(* CODESYS project HomePLC_AlarmManager.library
   Company: Tom Oyen
   Description: Alarm manager
   Version: 1.0
   Placeholder: HomePLC Alarm Manager
   Author: Tom Oyen
   Title: HomePLC Alarm Manager

Project tree, tasks and I/O mapping:
  libraries: HomePLC DIO, * (Tom Oyen); HomePLC General, * (Tom Oyen); HomePLC Logging, * (Tom Oyen); Tc2_Standard, * (Beckhoff Automation GmbH); Tc2_System, * (Beckhoff Automation GmbH); Tc3_Module, * (Beckhoff Automation GmbH)
  DUTs/
    data type E_AlarmManagerStep
    data type E_AlarmState
    data type ST_AlarmManagerHMI
  GVLs/
    global variables GVL_AlarmManager
  POUs/
    Keypad/
      DUTs/
        data type E_KeypadState
        data type ST_AlarmKeypadHMI
        data type ST_AlarmKeypadVirtual
        data type ST_LedState
      function block FB_AlarmKeypad [ST]: CheckCode, CollectInput, Execute, FB_init, Reset, SetAlarmState, SetBuzzer, SetConfiguredCode, SetLeds, UpdateHMI, HmiData, Name
      interface I_AlarmKeypad: CheckCode, Execute, SetAlarmState, SetBuzzer, SetConfiguredCode, HmiData, Name
    Sensor/
      DUTs/
        data type ST_AlarmSensorHMI
      function block FB_AlarmSensor [ST]: Execute, FB_init, UpdateHMI, Alarm, AlarmTrigger, HmiData, Tamper, TamperTrigger, WarnFirst
      interface I_AlarmSensor: Execute, Alarm, AlarmTrigger, HmiData, Tamper, TamperTrigger, WarnFirst
    Siren/
      DUTs/
        data type ST_AlarmSirenHMI
      function block FB_AlarmSiren [ST]: Execute, FB_init, SetLight, SetSound, UpdateHMI, HmiData, Tamper, TamperTrigger
      interface I_AlarmSiren: Execute, SetLight, SetSound, HmiData, Tamper, TamperTrigger
    function block FB_AlarmManager [ST]: AddKeypad, AddSensor, AddSiren, Execute, Execute_Keypads, Execute_Sensors, Execute_Sirens, FB_init, UpdateHMI
    interface I_AlarmManager: AddKeypad, AddSensor, AddSiren
  Project Information/
    function F_GetCompany [ST]
    function F_GetTitle [ST]
    function F_GetVersion [ST]
  Version/
    global variables Global_Version
  VISUs/
    visualisation Alarm
    visualisation Keypad
    visualisation Sensor
    visualisation Siren
  text list GlobalTextList
*)

// DUTs/E_AlarmManagerStep
{attribute 'qualified_only'}
{attribute 'strict'}
TYPE E_AlarmManagerStep :
(
	Init 					:= 0,
	CheckEnable				:= 1,
	
	HardwareCheck			:= 10,
	Enabling				:= 11,
	Enable					:= 12,
	
	CheckSensors			:= 20,
	
	Warn					:= 30,
	WaitForDisableWarn		:= 31,
	SoundAlarm				:= 32,
	WaitForDisableAlarm		:= 33,
	
	DisableAlarm			:= 40,
	
	Reset					:= 50
);
END_TYPE

// DUTs/E_AlarmState
{attribute 'qualified_only'}
{attribute 'strict'}
TYPE E_AlarmState :
(
	Off 			:= 0,
	Enabling		:= 1,
	On				:= 2
);
END_TYPE

// DUTs/ST_AlarmManagerHMI
TYPE ST_AlarmManagerHMI :
STRUCT
	// General
	nKeypads	: INT;		// Number of keypads
	nSensors	: INT;		// Number of sensors
	nSirens		: INT;		// Number of sirens
	bEnabled	: BOOL;		// Alarm enabled state
	
	// Overview
	aSensors	: ARRAY [0..GVL_AlarmManager.nMaxSensors - 1] OF ST_AlarmSensorHMI;
	aSirens		: ARRAY [0..GVL_AlarmManager.nMaxSirens - 1] OF ST_AlarmSirenHMI;
END_STRUCT
END_TYPE

// POUs/Keypad/DUTs/E_KeypadState
{attribute 'qualified_only'}
{attribute 'strict'}
TYPE E_KeypadState :
(
	Init 				:= 0,
	Idle				:= 1,
	InputDetected		:= 2,
	CheckInput			:= 3,
	Reset				:= 4	
);
END_TYPE

// POUs/Keypad/DUTs/ST_AlarmKeypadHMI
TYPE ST_AlarmKeypadHMI :
STRUCT
	sName			: STRING;
	
	bLed1			: BOOL;
	bLed2			: BOOL;
	bLed3			: BOOL;
	bLed4			: BOOL;
	bLed5			: BOOL;
	bLed6			: BOOL;
	
	bBuzzer			: BOOL;
	
	sCode			: STRING;
END_STRUCT
END_TYPE

// POUs/Keypad/DUTs/ST_AlarmKeypadVirtual
TYPE ST_AlarmKeypadVirtual :
STRUCT
	bButton1			: BOOL;
	bButton2			: BOOL;
	bButton3			: BOOL;
	bButton4			: BOOL;
	bButton5			: BOOL;
	bButton6			: BOOL;
END_STRUCT
END_TYPE

// POUs/Keypad/DUTs/ST_LedState
TYPE ST_LedState :
STRUCT
	eLed1	: E_DOCommand;
	eLed2	: E_DOCommand;
	eLed3	: E_DOCommand;
	eLed4	: E_DOCommand;
	eLed5	: E_DOCommand;
	eLed6	: E_DOCommand;
END_STRUCT
END_TYPE

// POUs/Sensor/DUTs/ST_AlarmSensorHMI
TYPE ST_AlarmSensorHMI :
STRUCT
	sName		: STRING;	// Sensor name
	bAlarm		: BOOL;		// True if the sensor detects something
	bTamper		: BOOL;		// True if the sensor is tampered with
END_STRUCT
END_TYPE

// POUs/Siren/DUTs/ST_AlarmSirenHMI
TYPE ST_AlarmSirenHMI :
STRUCT
	sName		: STRING;	// Siren name
	bSiren		: BOOL;		// True if the siren is on
	bLight		: BOOL;		// True if the light is on
	bTamper		: BOOL;		// True if the siren is tampered with
END_STRUCT
END_TYPE

// GVLs/GVL_AlarmManager
{attribute 'qualified_only'}
VAR_GLOBAL CONSTANT
	nMaxKeypads		: INT := 5;										// Maximum number of keypads
	nMaxSirens		: INT := 5;										// Maximum number of sirens
	nMaxSensors		: INT := 10;									// Maximum number of sensors
	sCode			: STRING := '1234';								// Configured alarm code
END_VAR

// Version/Global_Version
{attribute 'TcGenerated'}
{attribute 'no-analysis'}
{attribute 'linkalways'}
// This function has been automatically generated from the project information.
VAR_GLOBAL CONSTANT
	{attribute 'const_non_replaced'}
	stLibVersion_HomePLC_Alarm_Manager : ST_LibVersion := (iMajor := 1, iMinor := 0, iBuild := 0, iRevision := 0, nFlags := 0, sVersion := '1.0');
END_VAR

// POUs/Keypad/FB_AlarmKeypad
// Alarm keypad FB (B11-11-11L11-11-11)
FUNCTION_BLOCK FB_AlarmKeypad IMPLEMENTS I_AlarmKeypad
VAR
	sName			: STRING;				// Keypad name

	fbButton1		: FB_DigitalIn;			// Button 1
	fbLed1			: FB_DigitalOut;		// LED 1
	fbButton2		: FB_DigitalIn;			// Button 2
	fbLed2			: FB_DigitalOut;		// LED 2
	fbButton3		: FB_DigitalIn;			// Button 3
	fbLed3			: FB_DigitalOut;		// LED 3
	fbButton4		: FB_DigitalIn;			// Button 4
	fbLed4			: FB_DigitalOut;		// LED 4
	fbButton5		: FB_DigitalIn;			// Button 5
	fbLed5			: FB_DigitalOut;		// LED 5
	fbButton6		: FB_DigitalIn;			// Button 6
	fbLed6			: FB_DigitalOut;		// LED 6
	fbBuzzer		: FB_DigitalOut;		// Buzzer

	eState			: E_KeypadState;		// Keypad state
	sConfiguredCode	: STRING;				// Configured alarm code
	sInputCode		: STRING;				// User input code
	dtInputTime		: DATE_AND_TIME;		// Date and time of last user input
	stLedsDefault	: ST_LedState;			// Default LEDs state
	
	stHMI			: ST_AlarmKeypadHMI;	// HMI data
	stVirtual		: ST_AlarmKeypadVirtual;	// Virtual keypad
END_VAR

// Returns true if the user input code equals the configured code
METHOD CheckCode : BOOL
// Compare codes
CheckCode := sInputCode = sConfiguredCode;

// Reset input if correct code was entered
IF CheckCode THEN
	Reset();
END_IF
END_METHOD

// Collect user input from buttons and build the entered code, returns true if input was detected
METHOD PRIVATE CollectInput: BOOL
VAR
	sInput			: STRING;
END_VAR
// Check buttons and translate to input
IF fbButton1.Command = E_DICommand.ShortPress THEN sInput := '1'; END_IF
IF fbButton2.Command = E_DICommand.ShortPress THEN sInput := '2'; END_IF
IF fbButton3.Command = E_DICommand.ShortPress THEN sInput := '3'; END_IF
IF fbButton4.Command = E_DICommand.ShortPress THEN sInput := '4'; END_IF
IF fbButton5.Command = E_DICommand.ShortPress THEN sInput := '5'; END_IF
IF fbButton6.Command = E_DICommand.ShortPress THEN sInput := '6'; END_IF

// Check if input was detected
IF sInput <> '' THEN
	// Build user input code
	sInputCode := CONCAT(sInputCode, sInput);
	
	// Update time of last input
	dtInputTime := GetDateTime();
	
	// Set output
	CollectInput := TRUE;
ELSE
	// Set output
	CollectInput := FALSE;
END_IF
END_METHOD

// Run this method every cycle
METHOD Execute
VAR CONSTANT
	stLedsOn	: ST_LedState := (eLed1 := E_DOCommand.On,
									eLed2 := E_DOCommand.On,
									eLed3 := E_DOCommand.On,
									eLed4 := E_DOCommand.On,
									eLed5 := E_DOCommand.On,
									eLed6 := E_DOCommand.On);
END_VAR
// Keypad state machine
CASE eState OF
	E_KeypadState.Init:
		// Initialize
		eState := E_KeypadState.Idle;
	
	E_KeypadState.Idle:
		// Wait for input
		IF CollectInput() THEN
			eState := E_KeypadState.InputDetected;
		END_IF
	
	E_KeypadState.InputDetected:
		// Collect input in every state so no input is lost
		CollectInput();
		
		// Enable all LEDs
		SetLeds(stLedsOn);
		
		eState := E_KeypadState.CheckInput;
		
	E_KeypadState.CheckInput:
		// Continue collecting input
		CollectInput();
		
		// If no input is detected during some time, reset the keypad
		IF GetDateTime() - dtInputTime > T#2S THEN
			eState := E_KeypadState.Reset;
		END_IF
		
	E_KeypadState.Reset:
		// Reset keypad
		Reset();
		
		eState := E_KeypadState.Idle;
END_CASE

// Update HMI
UpdateHMI();
END_METHOD

METHOD FB_init : BOOL
VAR_INPUT
	bInitRetains	: BOOL;		// if TRUE, the retain variables are initialized (warm start / cold start)
	bInCopyCode		: BOOL;		// if TRUE, the instance afterwards gets moved into the copy code (online change)
	
	sKeypadName		: STRING;	// Keypad name
END_VAR
sName := sKeypadName;

fbBuzzer.SetBlinkPeriod(tPeriod := T#1500MS);
fbLed1.SetBlinkPeriod(tPeriod := T#1500MS);
END_METHOD

// Reset the keypad
METHOD PRIVATE Reset
// Reset user input code
sInputCode := '';

// Reset all LEDs to their default value
SetLeds(stLedsDefault);
END_METHOD

// Call this method once when the alarm state is changed
METHOD SetAlarmState
VAR_INPUT
	eAlarmState			: E_AlarmState;		// Alarm state
END_VAR
VAR CONSTANT
	stLedsAlarmOn		: ST_LedState := (eLed1 := E_DOCommand.On,
											eLed2 := E_DOCommand.Off,
											eLed3 := E_DOCommand.Off,
											eLed4 := E_DOCommand.Off,
											eLed5 := E_DOCommand.Off,
											eLed6 := E_DOCommand.Off);
	stLedsAlarmOff		: ST_LedState := (eLed1 := E_DOCommand.Off,
											eLed2 := E_DOCommand.Off,
											eLed3 := E_DOCommand.Off,
											eLed4 := E_DOCommand.Off,
											eLed5 := E_DOCommand.Off,
											eLed6 := E_DOCommand.Off);
	stLedsAlarmEnabling	: ST_LedState := (eLed1 := E_DOCommand.Blink,
											eLed2 := E_DOCommand.Off,
											eLed3 := E_DOCommand.Off,
											eLed4 := E_DOCommand.Off,
											eLed5 := E_DOCommand.Off,
											eLed6 := E_DOCommand.Off);
END_VAR
// Set LEDs default state
CASE eAlarmState OF
	E_AlarmState.Off:
		// Alarm is off
		stLedsDefault := stLedsAlarmOff;
		
	E_AlarmState.Enabling:
		// Alarm is enabling
		stLedsDefault := stLedsAlarmEnabling;
	
	E_AlarmState.On:
		// Alarm is on
		stLedsDefault := stLedsAlarmOn;
END_CASE

// Reset keypad
Reset();
END_METHOD

// Set the buzzer command
METHOD SetBuzzer
VAR_INPUT
	eCommand	: E_DOCommand;
END_VAR
// Set digital output command
fbBuzzer.SetCommand(eCommandIn := eCommand);
END_METHOD

// Set the keypad configured code
METHOD SetConfiguredCode
VAR_INPUT
	sCode	:	STRING;		// Configured code
END_VAR
// Set configured alarm code
sConfiguredCode := sCode;
END_METHOD

// Set the LEDs state
METHOD PRIVATE SetLeds
VAR_INPUT
	stLeds		: ST_LedState;		// LED states
END_VAR
fbLed1.SetCommand(eCommandIn := stLeds.eLed1);
fbLed2.SetCommand(eCommandIn := stLeds.eLed2);
fbLed3.SetCommand(eCommandIn := stLeds.eLed3);
fbLed4.SetCommand(eCommandIn := stLeds.eLed4);
fbLed5.SetCommand(eCommandIn := stLeds.eLed5);
fbLed6.SetCommand(eCommandIn := stLeds.eLed6);
END_METHOD

// Update HMI
METHOD PRIVATE UpdateHMI
VAR
	stLed1HMI	: ST_HmiDigitalOut;
	stLed2HMI	: ST_HmiDigitalOut;
	stLed3HMI	: ST_HmiDigitalOut;
	stLed4HMI	: ST_HmiDigitalOut;
	stLed5HMI	: ST_HmiDigitalOut;
	stLed6HMI	: ST_HmiDigitalOut;
	stBuzzerHMI	: ST_HmiDigitalOut;
END_VAR
// Get data
stLed1HMI := fbLed1.HmiData;
stLed2HMI := fbLed2.HmiData;
stLed3HMI := fbLed3.HmiData;
stLed4HMI := fbLed4.HmiData;
stLed5HMI := fbLed5.HmiData;
stLed6HMI := fbLed6.HmiData;
stBuzzerHMI := fbBuzzer.HmiData;

// Set HMI data
stHMI.bLed1 := stLed1HMI.bValue;
stHMI.bLed2 := stLed2HMI.bValue;
stHMI.bLed3 := stLed3HMI.bValue;
stHMI.bLed4 := stLed4HMI.bValue;
stHMI.bLed5 := stLed5HMI.bValue;
stHMI.bLed6 := stLed6HMI.bValue;
stHMI.bBuzzer := stBuzzerHMI.bValue;

stHMI.sCode := sInputCode;
stHMI.sName := sName;

// Set buttons
fbButton1.SetExternalIn(bIn := stVirtual.bButton1);
fbButton2.SetExternalIn(bIn := stVirtual.bButton2);
fbButton3.SetExternalIn(bIn := stVirtual.bButton3);
fbButton4.SetExternalIn(bIn := stVirtual.bButton4);
fbButton5.SetExternalIn(bIn := stVirtual.bButton5);
fbButton6.SetExternalIn(bIn := stVirtual.bButton6);
END_METHOD

// Returns the HMI data
PROPERTY HmiData : ST_AlarmKeypadHMI
GET
HmiData := stHMI;
END_GET
END_PROPERTY

// Returns the keypad name
PROPERTY Name : STRING
GET
Name := sName;
END_GET
END_PROPERTY

END_FUNCTION_BLOCK

// POUs/Keypad/I_AlarmKeypad
// Alarm keypad interface
INTERFACE I_AlarmKeypad

// Returns true if the user input code equals the configured code
METHOD CheckCode : BOOL
END_METHOD

// Run this method every cycle
METHOD Execute
END_METHOD

// Call this method once when the alarm state is changed
METHOD SetAlarmState
VAR_INPUT
	eAlarmState			: E_AlarmState;		// Alarm state
END_VAR
END_METHOD

// Set the buzzer command
METHOD SetBuzzer
VAR_INPUT
	eCommand	: E_DOCommand;
END_VAR
END_METHOD

// Set the keypad configured code
METHOD SetConfiguredCode
VAR_INPUT
	sCode	:	STRING;		// Configured code
END_VAR
END_METHOD

// Returns the HMI data
PROPERTY HmiData : ST_AlarmKeypadHMI
GET
END_GET
END_PROPERTY

// Returns the keypad name
PROPERTY Name : STRING
GET
END_GET
END_PROPERTY

END_INTERFACE

// POUs/Sensor/FB_AlarmSensor
// Alarm sensor FB
FUNCTION_BLOCK FB_AlarmSensor IMPLEMENTS I_AlarmSensor
VAR
	sName					: STRING;				// Sensor name
	bWarnFirst				: BOOL;					// Set to true to warn the user before setting off the alarm
	
	ibAlarm			AT %I*	: BOOL;					// Active low alarm input
	ibTamper		AT %I*	: BOOL;					// Active low tamper input
	
	bAlarm					: BOOL;					// True if the sensor detects something
	bTamper					: BOOL;					// True if the sensor is tampered with
	
	bAlarmTrigger			: BOOL;					// Returns true when the sensor is triggered
	bTamperTrigger			: BOOL;					// Returns true when the sensor is tampered with
	
	stHMI					: ST_AlarmSensorHMI;	// HMI data
END_VAR

// Run this method every cycle
METHOD Execute
VAR_INST
	fbAlarm		: R_TRIG;		// Alarm rising trigger
	fbTamper	: R_TRIG;		// Tamper rising trigger
END_VAR
// Convert active low inputs
bAlarm := NOT ibAlarm;
bTamper := NOT ibTamper;

// Run FBs
fbAlarm(CLK := bAlarm);
fbTamper(CLK := bTamper);

// Check triggers
bAlarmTrigger := fbAlarm.Q;
bTamperTrigger := fbTamper.Q;

// Update HMI
UpdateHMI();
END_METHOD

METHOD FB_init : BOOL
VAR_INPUT
	bInitRetains	: BOOL;		// if TRUE, the retain variables are initialized (warm start / cold start)
	bInCopyCode		: BOOL;		// if TRUE, the instance afterwards gets moved into the copy code (online change)
	
	sSensorName		: STRING;	// Sensor name
	bEnableWarning	: BOOL;		// Set to true to warn the user before setting off the alarm
END_VAR
sName := sSensorName;
bWarnFirst := bEnableWarning;
END_METHOD

// Update HMI
METHOD PRIVATE UpdateHMI
stHMI.sName := sName;
stHMI.bAlarm := bAlarm;
stHMI.bTamper := bTamper;
END_METHOD

// Returns true if the sensor detects something (as long as something is detected)
PROPERTY Alarm : BOOL
GET
Alarm := bAlarm;
END_GET
END_PROPERTY

// Returns true when the sensor is triggered (one cycle)
PROPERTY AlarmTrigger : BOOL
GET
AlarmTrigger := bAlarmTrigger;
END_GET
END_PROPERTY

// Returns the HMI data
PROPERTY HmiData : ST_AlarmSensorHMI
GET
HmiData := stHMI;
END_GET
END_PROPERTY

// Returns true when the sensor is tampered with (as long as the sensor is tampered with)
PROPERTY Tamper : BOOL
GET
Tamper := bTamper;
END_GET
END_PROPERTY

// Returns true when the tamper sensor is triggered (one cycle)
PROPERTY TamperTrigger : BOOL
GET
TamperTrigger := bTamperTrigger;
END_GET
END_PROPERTY

// Returs true if the user is warned before the alarm is set off
PROPERTY WarnFirst : BOOL
GET
WarnFirst := bWarnFirst;
END_GET
END_PROPERTY

END_FUNCTION_BLOCK

// POUs/Sensor/I_AlarmSensor
// Alarm sensor interface
INTERFACE I_AlarmSensor

// Run this method every cycle
METHOD Execute
END_METHOD

// Returns true if the sensor detects something (as long as something is detected)
PROPERTY Alarm : BOOL
GET
END_GET
END_PROPERTY

// Returns true when the sensor is triggered (one cycle)
PROPERTY AlarmTrigger : BOOL
GET
END_GET
END_PROPERTY

// Returns the HMI data
PROPERTY HmiData : ST_AlarmSensorHMI
GET
END_GET
END_PROPERTY

// Returns true when the sensor is tampered with (as long as the sensor is tampered with)
PROPERTY Tamper : BOOL
GET
END_GET
END_PROPERTY

// Returns true when the tamper sensor is triggered (one cycle)
PROPERTY TamperTrigger : BOOL
GET
END_GET
END_PROPERTY

// Returs true if the user is warned before the alarm is set off
PROPERTY WarnFirst : BOOL
GET
END_GET
END_PROPERTY

END_INTERFACE

// POUs/Siren/FB_AlarmSiren
// Alarm siren FB
FUNCTION_BLOCK FB_AlarmSiren IMPLEMENTS I_AlarmSiren
VAR
	sName				: STRING;				// Siren name
	
	ibTamper			AT %I* : BOOL;			// Active low tamper input
	fbLight				: FB_DigitalOut;		// Siren light digital output FB
	fbSiren				: FB_DigitalOut;		// Siren sound digital output FB
	
	bTamper				: BOOL;					// True if the siren is tampered with
	
	bTamperTrigger		: BOOL;					// True when the tamper sensor is triggered (one cycle)
	
	stHMI				: ST_AlarmSirenHMI;		// HMI data
END_VAR

// Run this method every cycle
METHOD Execute
VAR_INST
	fbTamper	: R_TRIG;		// Tamper rising edge
END_VAR
// Convert active low inputs
bTamper := NOT ibTamper;

// Run FBs
fbTamper(CLK := bTamper);

// Check trigger
bTamperTrigger := fbTamper.Q;

// Update HMI
UpdateHMI();
END_METHOD

METHOD FB_init : BOOL
VAR_INPUT
	bInitRetains	: BOOL;		// if TRUE, the retain variables are initialized (warm start / cold start)
	bInCopyCode		: BOOL;		// if TRUE, the instance afterwards gets moved into the copy code (online change)
	
	sSirenName		: STRING;	// Siren name
END_VAR
sName := sSirenName;
END_METHOD

// Set siren light
METHOD SetLight
VAR_INPUT
	eCommand	: E_DOCommand;		// Siren digital output command
END_VAR
// Set siren digital output command
fbLight.SetCommand(eCommandIn := eCommand);
END_METHOD

// Set siren sound
METHOD SetSound
VAR_INPUT
	eCommand	: E_DOCommand;		// Siren sound digital output command
END_VAR
// Set the siren digital output command
fbSiren.SetCommand(eCommandIn := eCommand);
END_METHOD

// Update HMI
METHOD PRIVATE UpdateHMI
VAR
	stSirenHMI	: ST_HmiDigitalOut;
	stLightHMI	: ST_HmiDigitalOut;
END_VAR
// Get data
stSirenHMI := fbSiren.HmiData;
stLightHMI := fbLight.HmiData;

// Set HMI data
stHMI.sName := sName;
stHMI.bSiren := stSirenHMI.bValue;
stHMI.bLight := stLightHMI.bValue;
stHMI.bTamper := bTamper;
END_METHOD

// Returns the HMI data
PROPERTY HmiData : ST_AlarmSirenHMI
GET
HmiData := stHMI;
END_GET
END_PROPERTY

// Returns true when the siren is tampered with (as long as the siren is tampered with)
PROPERTY Tamper : BOOL
GET
Tamper := bTamper;
END_GET
END_PROPERTY

// Returns true when the tamper sensor is triggered (one cycle)
PROPERTY TamperTrigger : BOOL
GET
TamperTrigger := bTamperTrigger;
END_GET
END_PROPERTY

END_FUNCTION_BLOCK

// POUs/Siren/I_AlarmSiren
INTERFACE I_AlarmSiren

// Run this method every cycle
METHOD Execute
END_METHOD

// Set siren light
METHOD SetLight
VAR_INPUT
	eCommand	: E_DOCommand;		// Siren digital output command
END_VAR
END_METHOD

// Set siren sound
METHOD SetSound
VAR_INPUT
	eCommand	: E_DOCommand;		// Siren sound digital output command
END_VAR
END_METHOD

// Returns the HMI data
PROPERTY HmiData : ST_AlarmSirenHMI
GET
END_GET
END_PROPERTY

// Returns true when the siren is tampered with (as long as the siren is tampered with)
PROPERTY Tamper : BOOL
GET
END_GET
END_PROPERTY

// Returns true when the tamper sensor is triggered (one cycle)
PROPERTY TamperTrigger : BOOL
GET
END_GET
END_PROPERTY

END_INTERFACE

// POUs/FB_AlarmManager
// Alarm manager
{attribute 'reflection'} 
FUNCTION_BLOCK FB_AlarmManager IMPLEMENTS I_AlarmManager
VAR
	aKeypads	: ARRAY [0..GVL_AlarmManager.nMaxKeypads - 1] OF I_AlarmKeypad;		// Keypads
	nKeypads	: INT;																// Number of keypads
	
	aSensors	: ARRAY [0..GVL_AlarmManager.nMaxSensors - 1] OF I_AlarmSensor;		// Alarm sensors
	nSensors	: INT;																// Number of alarm sensors
	
	aSirens		: ARRAY [0..GVL_AlarmManager.nMaxSirens - 1] OF I_AlarmSiren;		// Alarm sirens
	nSirens		: INT;																// Number of alarm sirens
	
	eState		: E_AlarmState;														// Alarm state
	
	fbLogger	: class_Tc3EventLogger;												// Logging FB

	// Use attributes to copy instance name to sName
	{attribute 'instance-path'} 
    {attribute 'noinit'} 
    sName		: STRING; 															// Instance name
	
	stHMI		: ST_AlarmManagerHMI;												// HMI data
END_VAR

// Add a keypad to the alarm manager
METHOD AddKeypad
VAR_INPUT
	IKeypad		: I_AlarmKeypad;		// Keypad interface
END_VAR
// Add keypad
aKeypads[nKeypads] := IKeypad;
nKeypads := nKeypads + 1;
END_METHOD

// Add an alarm sensor to the alarm manager
METHOD AddSensor
VAR_INPUT
	ISensor		: I_AlarmSensor;		// Alarm sensor interface
END_VAR
// Add alarm sensor
aSensors[nSensors] := ISensor;
nSensors := nSensors + 1;
END_METHOD

// Add a siren to the alarm manager
METHOD AddSiren
VAR_INPUT
	ISiren		: I_AlarmSiren;		// Siren interface
END_VAR
// Add siren
aSirens[nSirens] := ISiren;
nSirens := nSirens + 1;
END_METHOD

// Run this method every cycle
METHOD Execute
VAR_INST
	eStep						: E_AlarmManagerStep;		// Alarm manager state machine step
	eStepPrev					: E_AlarmManagerStep;		// Alarm manager state machine previous step
	bFirstCall					: BOOL;				// Alarm manager state machine step first call
	
	bCodeEntered				: BOOL;				// True if the configured code was entered on a keypad
	bSensorTriggered			: BOOL;				// True if a sensor is triggered
	bSensorTampered				: BOOL;				// True if a sensor is tampered with
	bWarn						: BOOL;				// True if the user needs to be warned first when a sensor is triggered
	bSirenTampered				: BOOL;				// True if a siren is tampered with
	
	eBuzzerCommand				: E_DOCommand;		// Keypad buzzer digital output command
	eSirenLightCommand			: E_DOCommand;		// Siren light digital output command
	eSirenSoundCommand			: E_DOCommand;		// Siren sound digital output command
	
	fbTimer						: TON;				// Timer FB
END_VAR
// Execute methods
Execute_Keypads(eBuzzerCommand := eBuzzerCommand,
				bCodeEntered => bCodeEntered);
Execute_Sensors(bSensorTriggered => bSensorTriggered,
				bSensorTampered => bSensorTampered,
				bWarn => bWarn);
Execute_Sirens(eLightCommand := eSirenLightCommand,
				eSoundCommand := eSirenSoundCommand,
				bSirenTampered => bSirenTampered);

// Set variables
bFirstCall := eStep <> eStepPrev;
eStepPrev := eStep;

// Execute alarm logic
CASE eStep OF
	E_AlarmManagerStep.Init:
		// Initialize
		eStep := E_AlarmManagerStep.CheckEnable;
		
	E_AlarmManagerStep.CheckEnable:
		// Check if configured code is entered by the user
		IF bCodeEntered THEN
			eStep := E_AlarmManagerStep.HardwareCheck;
		END_IF
		
	E_AlarmManagerStep.HardwareCheck:
		// Hardware check before enabling alarm
		
		// Check if a sensor detects something or if one is tampered with
		// Check if a siren is tampered with
		IF bSensorTampered OR bSirenTampered THEN
			// Sound buzzer to indicate alarm cannot be enabled
			eBuzzerCommand := E_DOCommand.Flash;
			
			fbLogger.AddInfo('Alarm cannot be enabled due to tampering');
			
			eStep := E_AlarmManagerStep.Reset;
		ELSE
			eStep := E_AlarmManagerStep.Enabling;
		END_IF
		
	E_AlarmManagerStep.Enabling:
		// Enabling alarm
		IF bFirstCall THEN
			// Initialize timer
			fbTimer.PT := T#20S;
			fbTimer(IN := FALSE);
			
			// Set alarm state
			eState := E_AlarmState.Enabling;
			
			// Set buzzer to blinking
			eBuzzerCommand := E_DOCommand.Blink;
		ELSE
			// Run timer FB
			fbTimer(IN := TRUE);
			
			// Check if timer expired
			IF fbTimer.Q THEN
				// Turn off buzzer
				eBuzzerCommand := E_DOCommand.Off;
			
				eStep := E_AlarmManagerStep.Enable;
			END_IF
		END_IF
	
	E_AlarmManagerStep.Enable:
		// Enable alarm
		eState := E_AlarmState.On;
		
		fbLogger.AddInfo('Alarm enabled');
		
		eStep := E_AlarmManagerStep.CheckSensors;
		
	E_AlarmManagerStep.CheckSensors:
		// Check if configure code is entered by user
		IF bCodeEntered THEN
			eStep := E_AlarmManagerStep.DisableAlarm;
		END_IF
		
		// Check if a sensor or siren is tampered with
		IF bSensorTampered OR bSirenTampered THEN
			eStep := E_AlarmManagerStep.SoundAlarm;
		END_IF
		
		// Check if a sensor detects something
		IF bSensorTriggered THEN
			// Check if user needs to be warned
			IF bWarn THEN
				eStep := E_AlarmManagerStep.Warn;
			ELSE
				eStep := E_AlarmManagerStep.SoundAlarm;
			END_IF
		END_IF
		
	E_AlarmManagerStep.Warn:
		// Warn the user before sounding the alarm
		eBuzzerCommand := E_DOCommand.On;
		
		fbLogger.AddInfo('Sensor triggered, warning user');
		
		eStep := E_AlarmManagerStep.WaitForDisableWarn;
		
	E_AlarmManagerStep.WaitForDisableWarn:
		// Wait for user to disable alarm and sound the alarm if it does not happen in time
		IF bFirstCall THEN
			// Initialize timer
			fbTimer.PT := T#30S;
			fbTimer(IN := FALSE);
		ELSE
			// Run timer FB
			fbTimer(IN := TRUE);
			
			// Check if configured code is entered by user
			IF bCodeEntered THEN
				// Disable alarm
				eStep := E_AlarmManagerStep.DisableAlarm;
			END_IF
			
			// Check if timer expired
			IF fbTimer.Q THEN
				// Sound alarm
				eStep := E_AlarmManagerStep.SoundAlarm;
			END_IF
		END_IF
		
	E_AlarmManagerStep.SoundAlarm:
		// Turn on alarm light and sound
		eSirenLightCommand := E_DOCommand.On;
		eSirenSoundCommand := E_DOCommand.On;
		
		// Turn off buzzer (if on)
		eBuzzerCommand := E_DOCommand.Off;
		
		fbLogger.AddInfo('Sounding alarm');
		
		eStep := E_AlarmManagerStep.WaitForDisableAlarm;
		
	E_AlarmManagerStep.WaitForDisableAlarm:
		// Wait for user to disable alarm or wait some time before turning it off automatically
		IF bFirstCall THEN
			// Initialize timer
			fbTimer.PT := T#3M;
			fbTimer(IN := FALSE);
		ELSE
			// Run timer FB
			fbTimer(IN := TRUE);
			
			// Check if configured code is entered by user or if timer expired
			IF bCodeEntered OR fbTimer.Q THEN
				// Disable alarm
				eStep := E_AlarmManagerStep.DisableAlarm;
			END_IF
		END_IF
		
	E_AlarmManagerStep.DisableAlarm:
		// Turn off alarm light and sounds
		eSirenLightCommand := E_DOCommand.Off;
		eSirenSoundCommand := E_DOCommand.Off;
		
		// Turn off buzzer (if on)
		eBuzzerCommand := E_DOCommand.Off;
		
		fbLogger.AddInfo('Alarm disabled');
		
		// Set alarm status
		eState := E_AlarmState.Off;
		
		eStep := E_AlarmManagerStep.Reset;
		
	E_AlarmManagerStep.Reset:
		eStep := E_AlarmManagerStep.CheckEnable;
		
END_CASE

// Update HMI
UpdateHMI();
END_METHOD

// Run this method every cycle
METHOD PRIVATE Execute_Keypads
VAR_INPUT
	eBuzzerCommand			: E_DOCommand;	// Keypad buzzer command
END_VAR
VAR_OUTPUT
	bCodeEntered			: BOOL;			// Returns true if the configured code is entered by the user
END_VAR
VAR_INST
	bInit					: BOOL;			// Initialized flag
	eBuzzerCommandPrev		: E_DOCommand;	// Previous buzzer digital output command
	fbBuzzerCommandTrigger	: R_TRIG;		// Buzzer command trigger
	eStatePrev				: E_AlarmState;	// Previous alarm state
	fbStateTrigger			: R_TRIG;		// Alarm state change trigger
END_VAR
VAR
	i						: INT;			// Iterator variable
END_VAR
// Check if buzzer command changed
fbBuzzerCommandTrigger(CLK := eBuzzerCommand <> eBuzzerCommandPrev);
eBuzzerCommandPrev := eBuzzerCommand;

// Check if alarm state changed
fbStateTrigger(CLK := eState <> eStatePrev);
eStatePrev := eState;

// Initialize variable
bCodeEntered := FALSE;

FOR i := 0 TO nKeypads - 1 DO	
	// Set keypad configure code
	aKeypads[i].SetConfiguredCode(sCode := GVL_AlarmManager.sCode);
	
	// Check if buzzer command changed
	IF fbBuzzerCommandTrigger.Q THEN
		// Set buzzer digital output command
		aKeypads[i].SetBuzzer(eCommand := eBuzzerCommand);
	END_IF
	
	// Check if alarm state changed
	IF fbStateTrigger.Q OR NOT bInit THEN
		// Update keypad on alarm state change
		aKeypads[i].SetAlarmState(eAlarmState := eState);
	END_IF
	
	// Run keypad Execute method
	aKeypads[i].Execute();
	
	// Check if the configured code is entered on at least one keypad
	bCodeEntered := bCodeEntered OR aKeypads[i].CheckCode();
END_FOR

bInit := TRUE;
END_METHOD

// Run this method every cycle
METHOD PRIVATE Execute_Sensors
VAR_OUTPUT
	bSensorTriggered	: BOOL;		// Returns true if a sensor detects something
	bSensorTampered		: BOOL;		// Returns true if a sensor is tampered with
	bWarn				: BOOL;		// Returns true if a warning is issued first instead of immediately sounding the alarm (only valid on sensor trigger)
END_VAR
VAR
	i					: INT;		// Iterator variable
END_VAR
// Initialize variables
bSensorTriggered := FALSE;
bSensorTampered	:= FALSE;
bWarn := TRUE;

FOR i := 0 TO nSensors -1 DO
	// Run sensor Execute method
	aSensors[i].Execute();

	// Check if at least one sensor detects something or is tampered with
	bSensorTriggered := bSensorTriggered OR aSensors[i].AlarmTrigger;
	bSensorTampered := bSensorTampered OR aSensors[i].TamperTrigger;
	
	// Check if alarm needs to be sounded immediately or if a warning can be issued first
	IF aSensors[i].AlarmTrigger AND NOT aSensors[i].TamperTrigger THEN
		// Sensor detects something but is not tampered with
		// Warn if the sensor allows a warning
		// If one sensor does not allow a warning, sound the alarm immediately
		bWarn := bWarn AND aSensors[i].WarnFirst;
	END_IF
END_FOR
END_METHOD

// Run this method every cycle
METHOD PRIVATE Execute_Sirens
VAR_INPUT
	eLightCommand				: E_DOCommand;		// Siren light digital output command
	eSoundCommand				: E_DOCommand;		// Siren sound digital output command
END_VAR
VAR_OUTPUT
	bSirenTampered				: BOOL;				// Returns true if the siren is tampered with
END_VAR
VAR
	i							: INT;				// Iterator variable
END_VAR
VAR_INST
	eLightCommandPrev			: E_DOCommand;		// Siren light previous digital output command
	fbLightCommandTrigger		: R_TRIG;			// Siren light command changed trigger
	
	eSoundCommandPrev			: E_DOCommand;		// Siren sound previous digital output command
	fbSoundCommandTrigger		: R_TRIG;			// Siren sound command changed trigger
END_VAR
// Check if the siren light digital command has changed
fbLightCommandTrigger(CLK := eLightCommand <> eLightCommandPrev);
eLightCommandPrev := eLightCommand;

// Check if the siren sound digital command has changed
fbSoundCommandTrigger(CLK := eSoundCommand <> eSoundCommandPrev);
eSoundCommandPrev := eSoundCommand;

// Initialize variable
bSirenTampered	:= FALSE;

FOR i := 0 TO nSirens - 1 DO
	// Check if siren light command changed
	IF fbLightCommandTrigger.Q THEN
		// Set siren light digital output command
		aSirens[i].SetLight(eCommand := eLightCommand);
	END_IF
	
	// Check if siren sound command changed
	IF fbSoundCommandTrigger.Q THEN
		// Set siren sound digital output command
		aSirens[i].SetSound(eCommand := eSoundCommand);
	END_IF
	
	// Run siren Execute method
	aSirens[i].Execute();
	
	// Check if at least one siren is tampered with
	bSirenTampered := bSirenTampered OR aSensors[i].TamperTrigger;
END_FOR
END_METHOD

// Initialize the alarm manager FB
METHOD FB_init : BOOL
VAR_INPUT
	bInitRetains : BOOL; // if TRUE, the retain variables are initialized (warm start / cold start)
	bInCopyCode : BOOL;  // if TRUE, the instance afterwards gets moved into the copy code (online change)
END_VAR
// Initialize logger
fbLogger.Init(sSource := sName, bEnableVerbose := TRUE);
END_METHOD

// Update HMI
METHOD PRIVATE UpdateHMI
VAR
	i	: INT;	// Iterator variable
END_VAR
// General
stHMI.nKeypads := nKeypads;
stHMI.nSensors := nSensors;
stHMI.nSirens := nSirens;
stHMI.bEnabled := eState = E_AlarmState.On;

// Overview
FOR i := 0 TO nSensors - 1 DO
	stHMI.aSensors[i] := aSensors[i].HmiData;
END_FOR

FOR i := 0 TO nSirens - 1 DO
	stHMI.aSirens[i] := aSirens[i].HmiData;
END_FOR
END_METHOD

END_FUNCTION_BLOCK

// POUs/I_AlarmManager
// Alarm manager interface
INTERFACE I_AlarmManager

// Add a keypad to the alarm manager
METHOD AddKeypad
VAR_INPUT
	IKeypad		: I_AlarmKeypad;		// Keypad interface
END_VAR
END_METHOD

// Add an alarm sensor to the alarm manager
METHOD AddSensor
VAR_INPUT
	ISensor		: I_AlarmSensor;		// Alarm sensor interface
END_VAR
END_METHOD

// Add a siren to the alarm manager
METHOD AddSiren
VAR_INPUT
	ISiren		: I_AlarmSiren;		// Siren interface
END_VAR
END_METHOD

END_INTERFACE

// Project Information/F_GetCompany
// This function has been automatically generated from the project information.
{attribute 'signature_flag' := '1073741824'}
{attribute 'TcGenerated'}
{attribute 'no-analysis'}
FUNCTION F_GetCompany : WSTRING
VAR_INPUT
	
END_VAR

F_GetCompany := "Tom Oyen";

END_FUNCTION

// Project Information/F_GetTitle
// This function has been automatically generated from the project information.
{attribute 'signature_flag' := '1073741824'}
{attribute 'TcGenerated'}
{attribute 'no-analysis'}
FUNCTION F_GetTitle : WSTRING
VAR_INPUT
	
END_VAR

F_GetTitle := "HomePLC Alarm Manager";

END_FUNCTION

// Project Information/F_GetVersion
// This function has been automatically generated from the project information.
{attribute 'signature_flag' := '1073741824'}
{attribute 'TcGenerated'}
{attribute 'no-analysis'}
FUNCTION F_GetVersion : ST_LibVersion
VAR_INPUT
	
END_VAR

F_GetVersion.iMajor := 1;
F_GetVersion.iMinor := 0;
F_GetVersion.iBuild := 0;
F_GetVersion.iRevision := 0;
F_GetVersion.sVersion := '1.0';
F_GetVersion.nFlags := 0;

END_FUNCTION

// VISUs/Alarm
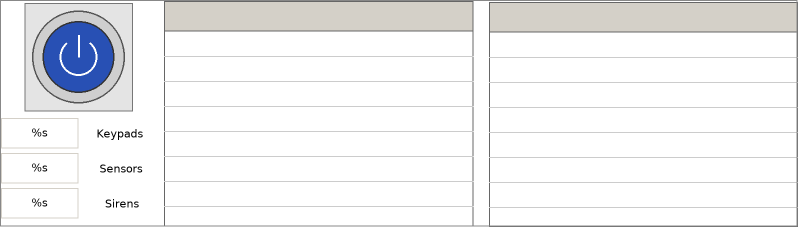
VISUALIZATION Alarm  // 798x227
VAR_IN_OUT
	stAlarm		: ST_AlarmManagerHMI;
END_VAR
    PowerSwitch (22,3 113x108), variable: stAlarm.bEnabled, input disabled if: TRUE, behaviour: TOGGLE, style: Switch-PowerSwitch-Blue
    Table (164,1 309x225), data array: stAlarm.aSensors
        p338671338: stAlarm.aSensors[INDEX].bTamper
        p3854506369: stAlarm.aSensors[INDEX].sName
        p1892666644: stAlarm.aSensors[INDEX].bAlarm
    Table (489,2 309x225), data array: stAlarm.aSirens
        p338671338: stAlarm.aSirens[INDEX].bLight
        p3854506369: stAlarm.aSirens[INDEX].sName
        p1892666644: stAlarm.aSirens[INDEX].bSiren
        p2170511999: stAlarm.aSirens[INDEX].bTamper
    Textfield (1,118 77x30), "%s", text variable: stAlarm.nKeypads
    Textfield (1,153 77x30), "%s", text variable: stAlarm.nSensors
    Textfield (1,188 77x30), "%s", text variable: stAlarm.nSirens
    Label (85,119 70x30), "Keypads"
    Label (86,154 70x30), "Sensors"
    Label (87,189 70x30), "Sirens"
END_VISUALIZATION

// VISUs/Keypad
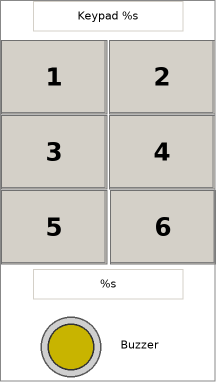
VISUALIZATION Keypad  // 216x382
VAR_IN_OUT
	stKeypadVirtual	: ST_AlarmKeypadVirtual;
	stKeypad		: ST_AlarmKeypadHMI;
END_VAR
    Button (1,40 106x74), "1", colour toggle: stKeypad.bLed1
        tap stKeypadVirtual.bButton1
    Button (109,40 106x74), "2", colour toggle: stKeypad.bLed2
        tap stKeypadVirtual.bButton2
    Button (1,115 106x74), "3", colour toggle: stKeypad.bLed3
        tap stKeypadVirtual.bButton3
    Button (109,115 106x74), "4", colour toggle: stKeypad.bLed4
        tap stKeypadVirtual.bButton4
    Button (1,190 106x74), "5", colour toggle: stKeypad.bLed5
        tap stKeypadVirtual.bButton5
    Button (110,190 106x74), "6", colour toggle: stKeypad.bLed6
        tap stKeypadVirtual.bButton6
    Lamp1 (36,312 70x70), variable: stKeypad.bBuzzer, style: Lamp-Lamp1-Yellow
    Label (115,330 49x30), "Buzzer"
    Textfield (33,269 150x30), "%s", text variable: stKeypad.sCode
    Textfield (33,1 150x30), "Keypad %s", text variable: stKeypad.sName
END_VISUALIZATION

// VISUs/Sensor
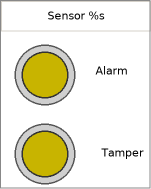
VISUALIZATION Sensor  // 151x189
VAR_IN_OUT
	stSensor		: ST_AlarmSensorHMI;
END_VAR
    Lamp1 (10,40 70x70), variable: stSensor.bAlarm, style: Lamp-Lamp1-Yellow
    Label (87,56 49x30), "Alarm"
    Textfield (1,1 150x30), "Sensor %s", text variable: stSensor.sName
    Lamp1 (10,119 70x70), variable: stSensor.bTamper, style: Lamp-Lamp1-Yellow
    Label (98,138 49x30), "Tamper"
END_VISUALIZATION

// VISUs/Siren
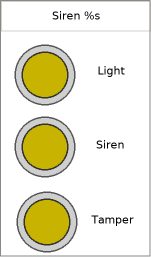
VISUALIZATION Siren  // 151x257
VAR_IN_OUT
	stSiren		: ST_AlarmSirenHMI;
END_VAR
    Lamp1 (10,40 70x70), variable: stSiren.bLight, style: Lamp-Lamp1-Yellow
    Lamp1 (10,112 70x70), variable: stSiren.bSiren, style: Lamp-Lamp1-Yellow
    Label (87,56 49x30), "Light"
    Label (86,130 49x30), "Siren"
    Textfield (1,1 150x30), "Siren %s", text variable: stSiren.sName
    Lamp1 (12,187 70x70), variable: stSiren.bTamper, style: Lamp-Lamp1-Yellow
    Label (88,205 49x30), "Tamper"
END_VISUALIZATION
